FUNCTION_BLOCK FB_Motor
VAR_INPUT
	bStart	: BOOL;
	bStop	: BOOL;
END_VAR
VAR_OUTPUT
	qMotor	: BOOL;
END_VAR
VAR
	
END_VAR

END_FUNCTION_BLOCK

(* stored: Version 1.1.0.1, ProductVersion 3.1.4024.11
   POU FB_Motor: Id {35ea3c71-53d6-4692-9667-037102dc0920}, SpecialFunc None *)
